(* PLC project Adressering.ecp, WAGO e!COCKPIT e!COCKPIT *)
(* stored: creationDateTime 2021-01-18T14:20:23.2110188, modificationDateTime 2021-01-18T11:51:27.6823754 *)

TYPE dtRomtype_22200000221102 : STRUCT
  RB601_V : BOOL;  (* Bevegelse *)
  RB602_V : BOOL;  (* Bevegelse *)
  RB601_HVAC : BOOL;  (* HVAC signal *)
  RB602_HVAC : BOOL;  (* HVAC signal *)
  RT601_CT : REAL;  (* Rom temperatur *)
  RT602_CT : REAL;  (* Rom temperatur *)
  RT602_SP : REAL;  (* Temperatur SP *)
  RT601_SP_D : REAL;  (* Temperatur SP *)
  RT601_SP_S : REAL;  (* Temperatur SP standby *)
  RT601_SP_N : REAL;  (* Temperatur SP nattsenk *)
  RT601_SP_F : REAL;  (* Temperatur SP frostsikring *)
  RT601_CS : REAL;  (* Aktivt temperatur SP *)
  OPM : INT;  (* Rom modus *)
  OPM_CV : INT;  (* Rom modus verdi *)
  RT601_SP : REAL;  (* Temperatur SP feedback *)
  RT601_SP_FB : REAL;  (* Temperatur SP *)
  RT601_SP_IN : REAL;  (* Temperatur SP lokalt panel *)
  RT602_SP_FB : REAL;  (* Temperatur SP *)
  RT602_SP_IN : REAL;  (* Temperatur SP lokalt panel *)
  LU601_V : BOOL;  (* Befukter status *)
  LU601_AL : BOOL;  (* Befukter alarm/feil *)
  OPM_001 : BYTE;  (* OPM output *)
  OPM_002 : BYTE;  (* OPM output *)
END_STRUCT;
END_TYPE

TYPE dtRomtype_1120011 : STRUCT
  RB601_V : BOOL;  (* Bevegelse *)
  RB601_HVAC : BOOL;  (* HVAC signal *)
  RT601_CT : REAL;  (* Rom temperatur *)
  RT602_CT : REAL;  (* Rom temperatur *)
  RT602_SP : REAL;  (* Temperatur SP *)
  RT601_SP_D : REAL;  (* Temperatur SP *)
  RT601_SP_S : REAL;  (* Temperatur SP standby *)
  RT601_SP_N : REAL;  (* Temperatur SP nattsenk *)
  RT601_SP_F : REAL;  (* Temperatur SP frostsikring *)
  RT601_CS : REAL;  (* Aktivt temperatur SP *)
  OPM : INT;  (* Rom modus *)
  OPM_CV : INT;  (* Rom modus verdi *)
  LH601_CMD : BOOL;  (* LH601_CMD *)
  LH601_MAN : BOOL;  (* Force LH *)
  LC601_OP : REAL;  (* LC601_OP *)
  LC601_SP : REAL;  (* LC SP *)
  LC601_MAN : BOOL;  (* Force LC *)
END_STRUCT;
END_TYPE

TYPE dtRomtype_112001 : STRUCT
  RB601_V : BOOL;  (* Bevegelse *)
  RB601_HVAC : BOOL;  (* HVAC signal *)
  RT601_CT : REAL;  (* Rom temperatur *)
  RT602_CT : REAL;  (* Rom temperatur *)
  RT602_SP : REAL;  (* Temperatur SP *)
  RT601_SP_D : REAL;  (* Temperatur SP *)
  RT601_SP_S : REAL;  (* Temperatur SP standby *)
  RT601_SP_N : REAL;  (* Temperatur SP nattsenk *)
  RT601_SP_F : REAL;  (* Temperatur SP frostsikring *)
  RT601_CS : REAL;  (* Aktivt temperatur SP *)
  OPM : INT;  (* Rom modus *)
  OPM_CV : INT;  (* Rom modus verdi *)
  LH601_CMD : BOOL;  (* LH601_CMD *)
  LH601_MAN : BOOL;  (* Force LH *)
END_STRUCT;
END_TYPE

TYPE dtRomtype_112101 : STRUCT
  RB601_V : BOOL;  (* Bevegelse *)
  RB601_HVAC : BOOL;  (* HVAC signal *)
  RT601_CT : REAL;  (* Rom temperatur *)
  RT602_CT : REAL;  (* Rom temperatur *)
  RT602_SP : REAL;  (* Temperatur SP *)
  RT601_SP_D : REAL;  (* Temperatur SP *)
  RT601_SP_S : REAL;  (* Temperatur SP standby *)
  RT601_SP_N : REAL;  (* Temperatur SP nattsenk *)
  RT601_SP_F : REAL;  (* Temperatur SP frostsikring *)
  RT601_CS : REAL;  (* Aktivt temperatur SP *)
  OPM : INT;  (* Rom modus *)
  OPM_CV : INT;  (* Rom modus verdi *)
  RY601_CV : REAL;  (* Co2 Nivaa *)
  RY601_SP : REAL;  (* Co2 SP *)
  RY601_OP : REAL;  (* Co2 paadrag *)
  LH601_CMD : BOOL;  (* LH601_CMD *)
  LH601_MAN : BOOL;  (* Force LH *)
END_STRUCT;
END_TYPE

TYPE dtRomtype_112002 : STRUCT
  RB601_V : BOOL;  (* Bevegelse *)
  RB601_HVAC : BOOL;  (* HVAC signal *)
  RT601_CT : REAL;  (* Rom temperatur *)
  RT602_CT : REAL;  (* Rom temperatur *)
  RT602_SP : REAL;  (* Temperatur SP *)
  RT601_SP_D : REAL;  (* Temperatur SP *)
  RT601_SP_S : REAL;  (* Temperatur SP standby *)
  RT601_SP_N : REAL;  (* Temperatur SP nattsenk *)
  RT601_SP_F : REAL;  (* Temperatur SP frostsikring *)
  RT601_CS : REAL;  (* Aktivt temperatur SP *)
  OPM : INT;  (* Rom modus *)
  OPM_CV : INT;  (* Rom modus verdi *)
  LH601_CMD : BOOL;  (* LH601_CMD *)
  LH602_CMD : BOOL;  (* LH602_CMD *)
  LH601_MAN : BOOL;  (* Force LH *)
END_STRUCT;
END_TYPE

TYPE dtRomtype_22 : STRUCT
  RB601_V : BOOL;  (* Bevegelse *)
  RB602_V : BOOL;  (* Bevegelse *)
  RB601_HVAC : BOOL;  (* HVAC signal *)
  RB602_HVAC : BOOL;  (* HVAC signal *)
END_STRUCT;
END_TYPE

TYPE dtRomtype_11 : STRUCT
  RB601_V : BOOL;  (* Bevegelse *)
  RB601_HVAC : BOOL;  (* HVAC signal *)
END_STRUCT;
END_TYPE

TYPE dtRomtype_4462051 : STRUCT
  RB601_V : BOOL;  (* Bevegelse *)
  RB602_V : BOOL;  (* Bevegelse *)
  RB603_V : BOOL;  (* Bevegelse *)
  RB604_V : BOOL;  (* Bevegelse *)
  RB601_HVAC : BOOL;  (* HVAC signal *)
  RB602_HVAC : BOOL;  (* HVAC signal *)
  RB603_HVAC : BOOL;  (* HVAC signal *)
  RB604_HVAC : BOOL;  (* HVAC signal *)
  RT601_CT : REAL;  (* Rom temperatur *)
  RT602_CT : REAL;  (* Rom temperatur *)
  RT602_SP : REAL;  (* Temperatur SP *)
  RT603_CT : REAL;  (* Rom temperatur *)
  RT603_SP : REAL;  (* Temperatur SP *)
  RT604_CT : REAL;  (* Rom temperatur *)
  RT604_SP : REAL;  (* Temperatur SP *)
  RT605_CT : REAL;  (* Rom temperatur *)
  RT605_SP : REAL;  (* Temperatur SP *)
  RT606_CT : REAL;  (* Rom temperatur *)
  RT606_SP : REAL;  (* Temperatur SP *)
  RT601_SP_D : REAL;  (* Temperatur SP *)
  RT601_SP_S : REAL;  (* Temperatur SP standby *)
  RT601_SP_N : REAL;  (* Temperatur SP nattsenk *)
  RT601_SP_F : REAL;  (* Temperatur SP frostsikring *)
  RT601_CS : REAL;  (* Aktivt temperatur SP *)
  OPM : INT;  (* Rom modus *)
  OPM_CV : INT;  (* Rom modus verdi *)
  RY601_CV : REAL;  (* Co2 Nivaa *)
  RY602_CV : REAL;  (* Co2 Nivaa *)
  RY601_SP : REAL;  (* Co2 SP *)
  RY601_OP : REAL;  (* Co2 paadrag *)
  LH601_CMD : BOOL;  (* LH601_CMD *)
  LH602_CMD : BOOL;  (* LH602_CMD *)
  LH603_CMD : BOOL;  (* LH603_CMD *)
  LH604_CMD : BOOL;  (* LH604_CMD *)
  LH605_CMD : BOOL;  (* LH605_CMD *)
  LH601_MAN : BOOL;  (* Force LH *)
  LC601_OP : REAL;  (* LC601_OP *)
  LC601_SP : REAL;  (* LC SP *)
  LC601_MAN : BOOL;  (* Force LC *)
END_STRUCT;
END_TYPE

TYPE dtRomtype_003 : STRUCT
  RT601_CT : REAL;  (* Rom temperatur *)
  RT602_CT : REAL;  (* Rom temperatur *)
  RT602_SP : REAL;  (* Temperatur SP *)
  RT603_CT : REAL;  (* Rom temperatur *)
  RT603_SP : REAL;  (* Temperatur SP *)
  RT601_SP_D : REAL;  (* Temperatur SP *)
  RT601_SP_S : REAL;  (* Temperatur SP standby *)
  RT601_SP_N : REAL;  (* Temperatur SP nattsenk *)
  RT601_SP_F : REAL;  (* Temperatur SP frostsikring *)
  RT601_CS : REAL;  (* Aktivt temperatur SP *)
  OPM : INT;  (* Rom modus *)
  OPM_CV : INT;  (* Rom modus verdi *)
END_STRUCT;
END_TYPE

TYPE dtRomtype_1121011 : STRUCT
  RB601_V : BOOL;  (* Bevegelse *)
  RB601_HVAC : BOOL;  (* HVAC signal *)
  RT601_CT : REAL;  (* Rom temperatur *)
  RT602_CT : REAL;  (* Rom temperatur *)
  RT602_SP : REAL;  (* Temperatur SP *)
  RT601_SP_D : REAL;  (* Temperatur SP *)
  RT601_SP_S : REAL;  (* Temperatur SP standby *)
  RT601_SP_N : REAL;  (* Temperatur SP nattsenk *)
  RT601_SP_F : REAL;  (* Temperatur SP frostsikring *)
  RT601_CS : REAL;  (* Aktivt temperatur SP *)
  OPM : INT;  (* Rom modus *)
  OPM_CV : INT;  (* Rom modus verdi *)
  RY601_CV : REAL;  (* Co2 Nivaa *)
  RY601_SP : REAL;  (* Co2 SP *)
  RY601_OP : REAL;  (* Co2 paadrag *)
  LH601_CMD : BOOL;  (* LH601_CMD *)
  LH601_MAN : BOOL;  (* Force LH *)
  LC601_OP : REAL;  (* LC601_OP *)
  LC601_SP : REAL;  (* LC SP *)
  LC601_MAN : BOOL;  (* Force LC *)
END_STRUCT;
END_TYPE

{attribute 'qualified_only'}
VAR_GLOBAL  (* STLV59_563 *)
  STLV59_A_563_RB001_HVAC : BOOL;  (* HVAC signal for PLS *)
  STLV59_A_563_KNX_Card_1_Status : BOOL;  (* KNX kort 1 status *)
  STLV59_A_563_001 : dtRomtype_22200000221102;  (* Ostelager *)
  STLV59_A_563_002 : dtRomtype_1120011;  (* Sosial sone *)
  STLV59_A_563_003 : dtRomtype_112001;  (* Jugendstue (Egentlig romtype 110001, men får temp fra rom 004) *)
  STLV59_A_563_004 : dtRomtype_112101;  (* Gang jugend *)
  STLV59_A_563_005 : dtRomtype_112001;  (* Kjøkken *)
  STLV59_A_563_006 : dtRomtype_112002;  (* Trenings rom *)
  STLV59_A_563_007 : dtRomtype_112001;  (* Garderobe 2 *)
  STLV59_A_563_008 : dtRomtype_112001;  (* Garderobe 1 *)
  STLV59_A_563_009 : dtRomtype_112001;  (* WC *)
  STLV59_A_563_010 : dtRomtype_112001;  (* WC *)
  STLV59_A_563_011 : dtRomtype_112001;  (* Garderobe *)
  STLV59_A_563_012 : dtRomtype_112001;  (* Entre *)
  STLV59_A_563_013 : dtRomtype_112001;  (* Bøttekott *)
  STLV59_A_563_014 : dtRomtype_22;  (* Teknisk rom *)
  STLV59_A_563_015 : dtRomtype_11;  (* Krypkjeller *)
  STLV59_A_563_016 : dtRomtype_11;  (* Teknisk rom tårn *)
  STLV59_A_563_017 : dtRomtype_112001;  (* Arkiv *)
  STLV59_A_563_101 : dtRomtype_112001;  (* Vindfang *)
  STLV59_A_563_102 : dtRomtype_112001;  (* Garderobe *)
  STLV59_A_563_103 : dtRomtype_4462051;  (* Storsal *)
  STLV59_A_563_109 : dtRomtype_112001;  (* Forrom WC *)
  STLV59_A_563_201 : dtRomtype_003;  (* Landskap *)
  STLV59_A_563_212 : dtRomtype_1121011;  (* Møterom 4 *)
  STLV59_A_563_213 : dtRomtype_1120011;  (* Stillerom *)
  STLV59_A_563_T1_U1 : dtRomtype_112001;  (* Trapp 1 U1 *)
  STLV59_A_563_T2_1 : dtRomtype_112001;  (* Trapp 2 1. etg. *)
  STLV59_A_563_T2_2 : dtRomtype_112001;  (* Trapp 2 2. etg. *)
END_VAR

FUNCTION_BLOCK fbRomtype_22200000221102
  VAR_INPUT
    RB601_HVAC : BOOL;
    RB602_HVAC : BOOL;
    RT601_CT : REAL;
    RT602_CT : REAL;
    RT602_SP : REAL;
    RT601_SP_D : REAL;
    RT601_SP_S : REAL;
    RT601_SP_N : REAL;
    RT601_SP_F : REAL;
    OPM : INT;
    RT601_SP_IN : REAL;
    RT602_SP_IN : REAL;
    LU601_V : BOOL;
  END_VAR
  VAR_OUTPUT
    OPM_CV : INT;
    RT601_CS : REAL;
    RT602_CS : REAL;
    OPM_001 : BYTE;
    OPM_002 : BYTE;
  END_VAR

(* CFC diagram, written out as Structured Text *)
END_FUNCTION_BLOCK

FUNCTION_BLOCK fbRomtype_1120011
  VAR_INPUT
    RB601_HVAC : BOOL;
    RT601_CT : REAL;
    RT602_CT : REAL;
    RT602_SP : REAL;
    RT601_SP_D : REAL;
    RT601_SP_S : REAL;
    RT601_SP_N : REAL;
    RT601_SP_F : REAL;
    OPM : INT;
    LH601_MAN : BOOL;
    LC601_SP : REAL;
    LC601_MAN : BOOL;
  END_VAR
  VAR_OUTPUT
    OPM_CV : INT;
    RT601_CS : REAL;
    RT602_CS : REAL;
    LH601_CMD : BOOL;
    LC601_OP : REAL;
  END_VAR

(* CFC diagram, written out as Structured Text *)
END_FUNCTION_BLOCK

FUNCTION_BLOCK fbRomtype_112001
  VAR_INPUT
    RB601_HVAC : BOOL;
    RT601_CT : REAL;
    RT602_CT : REAL;
    RT602_SP : REAL;
    RT601_SP_D : REAL;
    RT601_SP_S : REAL;
    RT601_SP_N : REAL;
    RT601_SP_F : REAL;
    OPM : INT;
    LH601_MAN : BOOL;
  END_VAR
  VAR_OUTPUT
    OPM_CV : INT;
    RT601_CS : REAL;
    RT602_CS : REAL;
    LH601_CMD : BOOL;
  END_VAR

(* CFC diagram, written out as Structured Text *)
END_FUNCTION_BLOCK

FUNCTION_BLOCK fbRomtype_112101
  VAR_INPUT
    RB601_HVAC : BOOL;
    RT601_CT : REAL;
    RT602_CT : REAL;
    RT602_SP : REAL;
    RT601_SP_D : REAL;
    RT601_SP_S : REAL;
    RT601_SP_N : REAL;
    RT601_SP_F : REAL;
    OPM : INT;
    RY601_CV : REAL;
    RY601_SP : REAL;
    LH601_MAN : BOOL;
  END_VAR
  VAR_OUTPUT
    OPM_CV : INT;
    RT601_CS : REAL;
    RT602_CS : REAL;
    RY601_OP : REAL;
    LH601_CMD : BOOL;
  END_VAR

(* CFC diagram, written out as Structured Text *)
END_FUNCTION_BLOCK

FUNCTION_BLOCK fbRomtype_112002
  VAR_INPUT
    RB601_HVAC : BOOL;
    RT601_CT : REAL;
    RT602_CT : REAL;
    RT602_SP : REAL;
    RT601_SP_D : REAL;
    RT601_SP_S : REAL;
    RT601_SP_N : REAL;
    RT601_SP_F : REAL;
    OPM : INT;
    LH601_MAN : BOOL;
  END_VAR
  VAR_OUTPUT
    OPM_CV : INT;
    RT601_CS : REAL;
    RT602_CS : REAL;
    LH601_CMD : BOOL;
    LH602_CMD : BOOL;
  END_VAR

(* CFC diagram, written out as Structured Text *)
END_FUNCTION_BLOCK

FUNCTION_BLOCK fbRomtype_4462051
  VAR_INPUT
    RB601_HVAC : BOOL;
    RB602_HVAC : BOOL;
    RB603_HVAC : BOOL;
    RB604_HVAC : BOOL;
    RT601_CT : REAL;
    RT602_CT : REAL;
    RT602_SP : REAL;
    RT603_CT : REAL;
    RT603_SP : REAL;
    RT604_CT : REAL;
    RT604_SP : REAL;
    RT605_CT : REAL;
    RT605_SP : REAL;
    RT606_CT : REAL;
    RT606_SP : REAL;
    RT601_SP_D : REAL;
    RT601_SP_S : REAL;
    RT601_SP_N : REAL;
    RT601_SP_F : REAL;
    OPM : INT;
    RY601_CV : REAL;
    RY602_CV : REAL;
    RY601_SP : REAL;
    LH601_MAN : BOOL;
    LC601_SP : REAL;
    LC601_MAN : BOOL;
  END_VAR
  VAR_OUTPUT
    OPM_CV : INT;
    RT601_CS : REAL;
    RT602_CS : REAL;
    RT603_CS : REAL;
    RT604_CS : REAL;
    RT605_CS : REAL;
    RT606_CS : REAL;
    RY601_OP : REAL;
    LH601_CMD : BOOL;
    LH602_CMD : BOOL;
    LH603_CMD : BOOL;
    LH604_CMD : BOOL;
    LH605_CMD : BOOL;
    LC601_OP : REAL;
  END_VAR

(* CFC diagram, written out as Structured Text *)
END_FUNCTION_BLOCK

FUNCTION_BLOCK fbRomtype_1121011
  VAR_INPUT
    RB601_HVAC : BOOL;
    RT601_CT : REAL;
    RT602_CT : REAL;
    RT602_SP : REAL;
    RT601_SP_D : REAL;
    RT601_SP_S : REAL;
    RT601_SP_N : REAL;
    RT601_SP_F : REAL;
    OPM : INT;
    RY601_CV : REAL;
    RY601_SP : REAL;
    LH601_MAN : BOOL;
    LC601_SP : REAL;
    LC601_MAN : BOOL;
  END_VAR
  VAR_OUTPUT
    OPM_CV : INT;
    RT601_CS : REAL;
    RT602_CS : REAL;
    RY601_OP : REAL;
    LH601_CMD : BOOL;
    LC601_OP : REAL;
  END_VAR

(* CFC diagram, written out as Structured Text *)
END_FUNCTION_BLOCK

PROGRAM PRG_KNX_563_1
  VAR
    i : INT := 0;  (* Felles *)
    Interval : OSCAT_BASIC.CLK_PRG;
    typDPT : typDPT;
    KNX_master_1 : WagoAppKNX.FbKNX_Master;  (* Master *)
    M1_001_001_RB601_V : fbDPT_Switch_pro;  (* 001 *)
    M1_002_001_RB602_V : fbDPT_Switch_pro;
    M1_003_001_RB601_HVAC : fbDPT_Switch_pro;
    M1_004_001_RB602_HVAC : fbDPT_Switch_pro;
    M1_005_001_RT601_SP : fbDPT_Value_Temp_pro;
    M1_006_001_RT602_SP : fbDPT_Value_Temp_pro;
    M1_007_001_RT601_SP_FB : fbDPT_Value_Temp_pro;
    M1_008_001_RT602_SP_FB : fbDPT_Value_Temp_pro;
    M1_009_001_OPM_001 : fbDPT_1_BYTE;
    M1_0010_001_OPM_002 : fbDPT_1_BYTE;
    M1_011_002_RB601_V : fbDPT_Switch_pro;  (* 002 *)
    M1_012_002_RB601_HVAC : fbDPT_Switch_pro;
    M1_013_002_RT601_CT : fbDPT_Value_Temp_pro;
    M1_014_002_RT602_CT : fbDPT_Value_Temp_pro;
    M1_015_003_RB601_V : fbDPT_Switch_pro;  (* 003 *)
    M1_016_003_RB601_HVAC : fbDPT_Switch_pro;
    M1_017_004_RB601_V : fbDPT_Switch_pro;  (* 004 *)
    M1_018_004_RB601_HVAC : fbDPT_Switch_pro;
    M1_019_004_RT601_CT : fbDPT_Value_Temp_pro;
    M1_020_004_RT602_CT : fbDPT_Value_Temp_pro;
    M1_021_004_RY601_CV : fbDPT_Value_AirQuality_pro;
    M1_022_005_RB601_V : fbDPT_Switch_pro;  (* 005 *)
    M1_023_005_RB601_HVAC : fbDPT_Switch_pro;
    M1_024_005_RT601_CT : fbDPT_Value_Temp_pro;
    M1_025_005_RT602_CT : fbDPT_Value_Temp_pro;
    M1_026_006_RB601_V : fbDPT_Switch_pro;  (* 006 *)
    M1_027_006_RB601_HVAC : fbDPT_Switch_pro;
    M1_028_006_RT601_CT : fbDPT_Value_Temp_pro;
    M1_029_007_RB601_V : fbDPT_Switch_pro;  (* 007 *)
    M1_030_007_RB601_HVAC : fbDPT_Switch_pro;
    M1_031_007_RT601_CT : fbDPT_Value_Temp_pro;
    M1_032_007_RT602_CT : fbDPT_Value_Temp_pro;
    M1_033_008_RB601_V : fbDPT_Switch_pro;  (* 008 *)
    M1_034_008_RB601_HVAC : fbDPT_Switch_pro;
    M1_035_008_RT601_CT : fbDPT_Value_Temp_pro;
    M1_036_008_RT602_CT : fbDPT_Value_Temp_pro;
    M1_037_009_RB601_V : fbDPT_Switch_pro;  (* 009 *)
    M1_038_009_RB601_HVAC : fbDPT_Switch_pro;
    M1_039_009_RT601_CT : fbDPT_Value_Temp_pro;
    M1_040_009_RT602_CT : fbDPT_Value_Temp_pro;
    M1_041_010_RB601_V : fbDPT_Switch_pro;  (* 010 *)
    M1_042_010_RB601_HVAC : fbDPT_Switch_pro;
    M1_043_010_RT601_CT : fbDPT_Value_Temp_pro;
    M1_044_010_RT602_CT : fbDPT_Value_Temp_pro;
    M1_045_011_RB601_V : fbDPT_Switch_pro;  (* 011 *)
    M1_046_011_RB601_HVAC : fbDPT_Switch_pro;
    M1_047_011_RT601_CT : fbDPT_Value_Temp_pro;
    M1_048_011_RT602_CT : fbDPT_Value_Temp_pro;
    M1_049_012_RB601_V : fbDPT_Switch_pro;  (* 012 *)
    M1_050_012_RB601_HVAC : fbDPT_Switch_pro;
    M1_051_012_RT601_CT : fbDPT_Value_Temp_pro;
    M1_052_012_RT602_CT : fbDPT_Value_Temp_pro;
    M1_053_013_RB601_V : fbDPT_Switch_pro;  (* 013 *)
    M1_054_013_RB601_HVAC : fbDPT_Switch_pro;
    M1_055_013_RT601_CT : fbDPT_Value_Temp_pro;
    M1_056_013_RT602_CT : fbDPT_Value_Temp_pro;
    M1_057_014_RB601_V : fbDPT_Switch_pro;  (* 014 *)
    M1_058_014_RB602_V : fbDPT_Switch_pro;
    M1_059_014_RB601_HVAC : fbDPT_Switch_pro;
    M1_060_014_RB602_HVAC : fbDPT_Switch_pro;
    M1_061_015_RB601_V : fbDPT_Switch_pro;  (* 015 *)
    M1_062_015_RB601_HVAC : fbDPT_Switch_pro;
    M1_063_016_RB601_V : fbDPT_Switch_pro;  (* 016 *)
    M1_064_016_RB601_HVAC : fbDPT_Switch_pro;
    M1_065_017_RB601_V : fbDPT_Switch_pro;  (* 017 *)
    M1_066_017_RB601_HVAC : fbDPT_Switch_pro;
    M1_067_017_RT601_CT : fbDPT_Value_Temp_pro;
    M1_068_017_RT602_CT : fbDPT_Value_Temp_pro;
    M1_069_101_RB601_V : fbDPT_Switch_pro;  (* 101 *)
    M1_070_101_RB601_HVAC : fbDPT_Switch_pro;
    M1_071_101_RT601_CT : fbDPT_Value_Temp_pro;
    M1_072_101_RT602_CT : fbDPT_Value_Temp_pro;
    M1_073_102_RB601_V : fbDPT_Switch_pro;  (* 102 *)
    M1_074_102_RB601_HVAC : fbDPT_Switch_pro;
    M1_075_102_RT601_CT : fbDPT_Value_Temp_pro;
    M1_076_102_RT602_CT : fbDPT_Value_Temp_pro;
    M1_077_103_RB601_V : fbDPT_Switch_pro;  (* 103 *)
    M1_078_103_RB602_V : fbDPT_Switch_pro;
    M1_079_103_RB603_V : fbDPT_Switch_pro;
    M1_080_103_RB604_V : fbDPT_Switch_pro;
    M1_081_103_RB601_HVAC : fbDPT_Switch_pro;
    M1_082_103_RB602_HVAC : fbDPT_Switch_pro;
    M1_083_103_RB603_HVAC : fbDPT_Switch_pro;
    M1_084_103_RB604_HVAC : fbDPT_Switch_pro;
    M1_085_103_RT601_CT : fbDPT_Value_Temp_pro;
    M1_086_103_RT602_CT : fbDPT_Value_Temp_pro;
    M1_087_103_RT603_CT : fbDPT_Value_Temp_pro;
    M1_088_103_RT604_CT : fbDPT_Value_Temp_pro;
    M1_089_109_RB601_V : fbDPT_Switch_pro;  (* 109 *)
    M1_090_109_RB601_HVAC : fbDPT_Switch_pro;
    M1_091_109_RT601_CT : fbDPT_Value_Temp_pro;
    M1_092_109_RT602_CT : fbDPT_Value_Temp_pro;
    M1_093_201_RT601_CT : fbDPT_Value_Temp_pro;  (* 201 *)
    M1_094_201_RT602_CT : fbDPT_Value_Temp_pro;
    M1_095_201_RT603_CT : fbDPT_Value_Temp_pro;
    M1_096_212_RB601_V : fbDPT_Switch_pro;  (* 212 *)
    M1_097_212_RB601_HVAC : fbDPT_Switch_pro;
    M1_098_212_RT601_CT : fbDPT_Value_Temp_pro;
    M1_099_212_RT602_CT : fbDPT_Value_Temp_pro;
    M1_100_212_RY601_CV : fbDPT_Value_AirQuality_pro;
    M1_101_213_RB601_V : fbDPT_Switch_pro;  (* 213 *)
    M1_102_213_RB601_HVAC : fbDPT_Switch_pro;
    M1_103_213_RT601_CT : fbDPT_Value_Temp_pro;
    M1_104_213_RT602_CT : fbDPT_Value_Temp_pro;
    M1_105_T1_U1_RB601_V : fbDPT_Switch_pro;  (* T1_U1 *)
    M1_106_T1_U1_RB601_HVAC : fbDPT_Switch_pro;
    M1_107_T1_U1_RT601_CT : fbDPT_Value_Temp_pro;
    M1_108_T1_U1_RT602_CT : fbDPT_Value_Temp_pro;
    M1_109_T2_1_RB601_V : fbDPT_Switch_pro;  (* T2_1 *)
    M1_110_T2_1_RB601_HVAC : fbDPT_Switch_pro;
    M1_111_T2_1_RT601_CT : fbDPT_Value_Temp_pro;
    M1_112_T2_1_RT602_CT : fbDPT_Value_Temp_pro;
    M1_113_T2_2_RB601_V : fbDPT_Switch_pro;  (* T2_2 *)
    M1_114_T2_2_RB601_HVAC : fbDPT_Switch_pro;
    M1_115_T2_2_RT601_CT : fbDPT_Value_Temp_pro;
    M1_116_T2_2_RT602_CT : fbDPT_Value_Temp_pro;
  END_VAR
  VAR  (* added by the conversion: wires and edge detectors of the diagram *)
    _ADD9_OUT : INT;
    _GT15_OUT : BOOL;
    _MOVE19_ENO : BOOL;
    _MOVE19_OUT : INT;
  END_VAR

(* CFC diagram, written out as Structured Text *)
(* KNX Sending interval *)
(* KNX Master *)
Interval(PT := t#2M);
_ADD9_OUT := BOOL_TO_INT(Interval.Q) + i;
i := _ADD9_OUT;
_GT15_OUT := i > 0;
_MOVE19_OUT := MOVE(EN := _GT15_OUT, IN := 0, ENO => _MOVE19_ENO);
IF _MOVE19_ENO THEN i := _MOVE19_OUT; END_IF;
KNX_master_1(I_Port := IoConfig_Globals.KNX_EIB_TP1_Interface, bPortKNX := 1);
STLV59_563.STLV59_A_563_KNX_Card_1_Status := KNX_master_1.sStatus = 'OK';
(* Rom 001 *)
(* RB601_V *)
(* RB602_V *)
M1_001_001_RB601_V(bPortKNX := 1, dwIndex_DPT := 1, typDPT := typDPT);
STLV59_563.STLV59_A_563_001.RB601_V := M1_001_001_RB601_V.xSwitch_OUT;
M1_002_001_RB602_V(bPortKNX := 1, dwIndex_DPT := 2, typDPT := typDPT);
STLV59_563.STLV59_A_563_001.RB602_V := M1_002_001_RB602_V.xSwitch_OUT;
(* RB601_HVAC *)
(* RB602_HVAC *)
M1_003_001_RB601_HVAC(bPortKNX := 1, dwIndex_DPT := 3, typDPT := typDPT);
STLV59_563.STLV59_A_563_001.RB601_HVAC := M1_003_001_RB601_HVAC.xSwitch_OUT;
M1_004_001_RB602_HVAC(bPortKNX := 1, dwIndex_DPT := 4, typDPT := typDPT);
STLV59_563.STLV59_A_563_001.RB602_HVAC := M1_004_001_RB602_HVAC.xSwitch_OUT;
(* RT601_SP *)
(* RT602_SP *)
M1_005_001_RT601_SP(bPortKNX := 1, dwIndex_DPT := 5, rValue_IN := STLV59_563.STLV59_A_563_001.RT601_SP_D, xUpdate_KNX := NOT STLV59_563.STLV59_A_563_001.RB601_HVAC, typDPT := typDPT);
M1_006_001_RT602_SP(bPortKNX := 1, dwIndex_DPT := 6, rValue_IN := STLV59_563.STLV59_A_563_001.RT602_SP, xUpdate_KNX := NOT STLV59_563.STLV59_A_563_001.RB601_HVAC, typDPT := typDPT);
(* RT601_SP Feedback *)
(* RT602_SP Feedback *)
M1_007_001_RT601_SP_FB(bPortKNX := 1, dwIndex_DPT := 7, typDPT := typDPT);
STLV59_563.STLV59_A_563_001.RT601_SP_IN := M1_007_001_RT601_SP_FB.rValue_OUT;
M1_008_001_RT602_SP_FB(bPortKNX := 1, dwIndex_DPT := 8, typDPT := typDPT);
STLV59_563.STLV59_A_563_001.RT602_SP_IN := M1_008_001_RT602_SP_FB.rValue_OUT;
(* OPM_001 *)
(* OPM_002 *)
M1_009_001_OPM_001(bPortKNX := 1, dwIndex_DPT := 9, bIN := STLV59_563.STLV59_A_563_001.OPM_001, xUpdate_KNX := i = 0, typDPT := typDPT);
M1_0010_001_OPM_002(bPortKNX := 1, dwIndex_DPT := 10, bIN := STLV59_563.STLV59_A_563_001.OPM_002, xUpdate_KNX := i = 1, typDPT := typDPT);
(* Rom 002 *)
(* RB601_V *)
(* RB601_HVAC *)
M1_011_002_RB601_V(bPortKNX := 1, dwIndex_DPT := 11, typDPT := typDPT);
STLV59_563.STLV59_A_563_002.RB601_V := M1_011_002_RB601_V.xSwitch_OUT;
M1_012_002_RB601_HVAC(bPortKNX := 1, dwIndex_DPT := 12, typDPT := typDPT);
STLV59_563.STLV59_A_563_002.RB601_HVAC := M1_012_002_RB601_HVAC.xSwitch_OUT;
(* RT601_CT *)
(* RT602_CT *)
M1_013_002_RT601_CT(bPortKNX := 1, dwIndex_DPT := 13, typDPT := typDPT);
STLV59_563.STLV59_A_563_002.RT601_CT := M1_013_002_RT601_CT.rValue_OUT;
M1_014_002_RT602_CT(bPortKNX := 1, dwIndex_DPT := 14, typDPT := typDPT);
STLV59_563.STLV59_A_563_002.RT602_CT := M1_014_002_RT602_CT.rValue_OUT;
(* Rom 003 *)
(* RB601_V *)
(* RB601_HVAC *)
M1_015_003_RB601_V(bPortKNX := 1, dwIndex_DPT := 15, typDPT := typDPT);
STLV59_563.STLV59_A_563_003.RB601_V := M1_015_003_RB601_V.xSwitch_OUT;
M1_016_003_RB601_HVAC(bPortKNX := 1, dwIndex_DPT := 16, typDPT := typDPT);
STLV59_563.STLV59_A_563_003.RB601_HVAC := M1_016_003_RB601_HVAC.xSwitch_OUT;
(* Rom 004 *)
(* RB601_V *)
(* RB601_HVAC *)
M1_017_004_RB601_V(bPortKNX := 1, dwIndex_DPT := 17, typDPT := typDPT);
STLV59_563.STLV59_A_563_004.RB601_V := M1_017_004_RB601_V.xSwitch_OUT;
M1_018_004_RB601_HVAC(bPortKNX := 1, dwIndex_DPT := 18, typDPT := typDPT);
STLV59_563.STLV59_A_563_004.RB601_HVAC := M1_018_004_RB601_HVAC.xSwitch_OUT;
(* RT601_CT *)
(* RT602_CT *)
M1_019_004_RT601_CT(bPortKNX := 1, dwIndex_DPT := 19, typDPT := typDPT);
STLV59_563.STLV59_A_563_004.RT601_CT := M1_019_004_RT601_CT.rValue_OUT;
M1_020_004_RT602_CT(bPortKNX := 1, dwIndex_DPT := 20, typDPT := typDPT);
STLV59_563.STLV59_A_563_004.RT602_CT := M1_020_004_RT602_CT.rValue_OUT;
(* RY601_CV *)
M1_021_004_RY601_CV(bPortKNX := 1, dwIndex_DPT := 21, typDPT := typDPT);
STLV59_563.STLV59_A_563_004.RY601_CV := M1_021_004_RY601_CV.rValue_OUT;
(* Rom 005 *)
(* RB601_V *)
(* RB601_HVAC *)
M1_022_005_RB601_V(bPortKNX := 1, dwIndex_DPT := 22, typDPT := typDPT);
STLV59_563.STLV59_A_563_005.RB601_V := M1_022_005_RB601_V.xSwitch_OUT;
M1_023_005_RB601_HVAC(bPortKNX := 1, dwIndex_DPT := 23, typDPT := typDPT);
STLV59_563.STLV59_A_563_005.RB601_HVAC := M1_023_005_RB601_HVAC.xSwitch_OUT;
(* RT601_CT *)
(* RT602_CT *)
M1_024_005_RT601_CT(bPortKNX := 1, dwIndex_DPT := 24, typDPT := typDPT);
STLV59_563.STLV59_A_563_005.RT601_CT := M1_024_005_RT601_CT.rValue_OUT;
M1_025_005_RT602_CT(bPortKNX := 1, dwIndex_DPT := 25, typDPT := typDPT);
STLV59_563.STLV59_A_563_005.RT602_CT := M1_025_005_RT602_CT.rValue_OUT;
(* Rom 006 *)
(* RB601_V *)
(* RB601_HVAC *)
M1_026_006_RB601_V(bPortKNX := 1, dwIndex_DPT := 26, typDPT := typDPT);
STLV59_563.STLV59_A_563_006.RB601_V := M1_026_006_RB601_V.xSwitch_OUT;
M1_027_006_RB601_HVAC(bPortKNX := 1, dwIndex_DPT := 27, typDPT := typDPT);
STLV59_563.STLV59_A_563_006.RB601_HVAC := M1_027_006_RB601_HVAC.xSwitch_OUT;
(* RT601_CT *)
M1_028_006_RT601_CT(bPortKNX := 1, dwIndex_DPT := 28, typDPT := typDPT);
STLV59_563.STLV59_A_563_006.RT601_CT := M1_028_006_RT601_CT.rValue_OUT;
(* Rom 007 *)
(* RB601_V *)
(* RB601_HVAC *)
M1_029_007_RB601_V(bPortKNX := 1, dwIndex_DPT := 29, typDPT := typDPT);
STLV59_563.STLV59_A_563_007.RB601_V := M1_029_007_RB601_V.xSwitch_OUT;
M1_030_007_RB601_HVAC(bPortKNX := 1, dwIndex_DPT := 30, typDPT := typDPT);
STLV59_563.STLV59_A_563_007.RB601_HVAC := M1_030_007_RB601_HVAC.xSwitch_OUT;
(* RT601_CT *)
(* RT602_CT *)
M1_031_007_RT601_CT(bPortKNX := 1, dwIndex_DPT := 31, typDPT := typDPT);
STLV59_563.STLV59_A_563_007.RT601_CT := M1_031_007_RT601_CT.rValue_OUT;
M1_032_007_RT602_CT(bPortKNX := 1, dwIndex_DPT := 32, typDPT := typDPT);
STLV59_563.STLV59_A_563_007.RT602_CT := M1_032_007_RT602_CT.rValue_OUT;
(* Rom 008 *)
(* RB601_V *)
(* RB601_HVAC *)
M1_033_008_RB601_V(bPortKNX := 1, dwIndex_DPT := 33, typDPT := typDPT);
STLV59_563.STLV59_A_563_008.RB601_V := M1_033_008_RB601_V.xSwitch_OUT;
M1_034_008_RB601_HVAC(bPortKNX := 1, dwIndex_DPT := 34, typDPT := typDPT);
STLV59_563.STLV59_A_563_008.RB601_HVAC := M1_034_008_RB601_HVAC.xSwitch_OUT;
(* RT601_CT *)
(* RT602_CT *)
M1_035_008_RT601_CT(bPortKNX := 1, dwIndex_DPT := 35, typDPT := typDPT);
STLV59_563.STLV59_A_563_008.RT601_CT := M1_035_008_RT601_CT.rValue_OUT;
M1_036_008_RT602_CT(bPortKNX := 1, dwIndex_DPT := 36, typDPT := typDPT);
STLV59_563.STLV59_A_563_008.RT602_CT := M1_036_008_RT602_CT.rValue_OUT;
(* Rom 009 *)
(* RB601_V *)
(* RB601_HVAC *)
M1_037_009_RB601_V(bPortKNX := 1, dwIndex_DPT := 37, typDPT := typDPT);
STLV59_563.STLV59_A_563_009.RB601_V := M1_037_009_RB601_V.xSwitch_OUT;
M1_038_009_RB601_HVAC(bPortKNX := 1, dwIndex_DPT := 38, typDPT := typDPT);
STLV59_563.STLV59_A_563_009.RB601_HVAC := M1_038_009_RB601_HVAC.xSwitch_OUT;
(* RT601_CT *)
(* RT602_CT *)
M1_039_009_RT601_CT(bPortKNX := 1, dwIndex_DPT := 39, typDPT := typDPT);
STLV59_563.STLV59_A_563_009.RT601_CT := M1_039_009_RT601_CT.rValue_OUT;
M1_040_009_RT602_CT(bPortKNX := 1, dwIndex_DPT := 40, typDPT := typDPT);
STLV59_563.STLV59_A_563_009.RT602_CT := M1_040_009_RT602_CT.rValue_OUT;
(* Rom 010 *)
(* RB601_V *)
(* RB601_HVAC *)
M1_041_010_RB601_V(bPortKNX := 1, dwIndex_DPT := 41, typDPT := typDPT);
STLV59_563.STLV59_A_563_010.RB601_V := M1_041_010_RB601_V.xSwitch_OUT;
M1_042_010_RB601_HVAC(bPortKNX := 1, dwIndex_DPT := 42, typDPT := typDPT);
STLV59_563.STLV59_A_563_010.RB601_HVAC := M1_042_010_RB601_HVAC.xSwitch_OUT;
(* RT601_CT *)
(* RT602_CT *)
M1_043_010_RT601_CT(bPortKNX := 1, dwIndex_DPT := 43, typDPT := typDPT);
STLV59_563.STLV59_A_563_010.RT601_CT := M1_043_010_RT601_CT.rValue_OUT;
M1_044_010_RT602_CT(bPortKNX := 1, dwIndex_DPT := 44, typDPT := typDPT);
STLV59_563.STLV59_A_563_010.RT602_CT := M1_044_010_RT602_CT.rValue_OUT;
(* Rom 011 *)
(* RB601_V *)
(* RB601_HVAC *)
M1_045_011_RB601_V(bPortKNX := 1, dwIndex_DPT := 45, typDPT := typDPT);
STLV59_563.STLV59_A_563_011.RB601_V := M1_045_011_RB601_V.xSwitch_OUT;
M1_046_011_RB601_HVAC(bPortKNX := 1, dwIndex_DPT := 46, typDPT := typDPT);
STLV59_563.STLV59_A_563_011.RB601_HVAC := M1_046_011_RB601_HVAC.xSwitch_OUT;
(* RT601_CT *)
(* RT602_CT *)
M1_047_011_RT601_CT(bPortKNX := 1, dwIndex_DPT := 47, typDPT := typDPT);
STLV59_563.STLV59_A_563_011.RT601_CT := M1_047_011_RT601_CT.rValue_OUT;
M1_048_011_RT602_CT(bPortKNX := 1, dwIndex_DPT := 48, typDPT := typDPT);
STLV59_563.STLV59_A_563_011.RT602_CT := M1_048_011_RT602_CT.rValue_OUT;
(* Rom 012 *)
(* RB601_V *)
(* RB601_HVAC *)
M1_049_012_RB601_V(bPortKNX := 1, dwIndex_DPT := 49, typDPT := typDPT);
STLV59_563.STLV59_A_563_012.RB601_V := M1_049_012_RB601_V.xSwitch_OUT;
M1_050_012_RB601_HVAC(bPortKNX := 1, dwIndex_DPT := 50, typDPT := typDPT);
STLV59_563.STLV59_A_563_012.RB601_HVAC := M1_050_012_RB601_HVAC.xSwitch_OUT;
(* RT601_CT *)
(* RT602_CT *)
M1_051_012_RT601_CT(bPortKNX := 1, dwIndex_DPT := 51, typDPT := typDPT);
STLV59_563.STLV59_A_563_012.RT601_CT := M1_051_012_RT601_CT.rValue_OUT;
M1_052_012_RT602_CT(bPortKNX := 1, dwIndex_DPT := 52, typDPT := typDPT);
STLV59_563.STLV59_A_563_012.RT602_CT := M1_052_012_RT602_CT.rValue_OUT;
(* Rom 013 *)
(* RB601_V *)
(* RB601_HVAC *)
M1_053_013_RB601_V(bPortKNX := 1, dwIndex_DPT := 53, typDPT := typDPT);
STLV59_563.STLV59_A_563_013.RB601_V := M1_053_013_RB601_V.xSwitch_OUT;
M1_054_013_RB601_HVAC(bPortKNX := 1, dwIndex_DPT := 54, typDPT := typDPT);
STLV59_563.STLV59_A_563_013.RB601_HVAC := M1_054_013_RB601_HVAC.xSwitch_OUT;
(* RT601_CT *)
(* RT602_CT *)
M1_055_013_RT601_CT(bPortKNX := 1, dwIndex_DPT := 55, typDPT := typDPT);
STLV59_563.STLV59_A_563_013.RT601_CT := M1_055_013_RT601_CT.rValue_OUT;
M1_056_013_RT602_CT(bPortKNX := 1, dwIndex_DPT := 56, typDPT := typDPT);
STLV59_563.STLV59_A_563_013.RT602_CT := M1_056_013_RT602_CT.rValue_OUT;
(* Rom 014 *)
(* RB601_V *)
(* RB602_V *)
M1_057_014_RB601_V(bPortKNX := 1, dwIndex_DPT := 57, typDPT := typDPT);
STLV59_563.STLV59_A_563_014.RB601_V := M1_057_014_RB601_V.xSwitch_OUT;
M1_058_014_RB602_V(bPortKNX := 1, dwIndex_DPT := 58, typDPT := typDPT);
STLV59_563.STLV59_A_563_014.RB602_V := M1_058_014_RB602_V.xSwitch_OUT;
(* RB601_HVAC *)
(* RB602_HVAC *)
M1_059_014_RB601_HVAC(bPortKNX := 1, dwIndex_DPT := 59, typDPT := typDPT);
STLV59_563.STLV59_A_563_014.RB601_HVAC := M1_059_014_RB601_HVAC.xSwitch_OUT;
M1_060_014_RB602_HVAC(bPortKNX := 1, dwIndex_DPT := 60, typDPT := typDPT);
STLV59_563.STLV59_A_563_014.RB602_HVAC := M1_060_014_RB602_HVAC.xSwitch_OUT;
(* Rom 015 *)
(* RB601_V *)
(* RB601_HVAC *)
M1_061_015_RB601_V(bPortKNX := 1, dwIndex_DPT := 61, typDPT := typDPT);
STLV59_563.STLV59_A_563_015.RB601_V := M1_061_015_RB601_V.xSwitch_OUT;
M1_062_015_RB601_HVAC(bPortKNX := 1, dwIndex_DPT := 62, typDPT := typDPT);
STLV59_563.STLV59_A_563_015.RB601_HVAC := M1_062_015_RB601_HVAC.xSwitch_OUT;
(* Rom 016 *)
(* RB601_V *)
(* RB601_HVAC *)
M1_063_016_RB601_V(bPortKNX := 1, dwIndex_DPT := 63, typDPT := typDPT);
STLV59_563.STLV59_A_563_016.RB601_V := M1_063_016_RB601_V.xSwitch_OUT;
M1_064_016_RB601_HVAC(bPortKNX := 1, dwIndex_DPT := 64, typDPT := typDPT);
STLV59_563.STLV59_A_563_016.RB601_HVAC := M1_064_016_RB601_HVAC.xSwitch_OUT;
(* Rom 017 *)
(* RB601_V *)
(* RB601_HVAC *)
M1_065_017_RB601_V(bPortKNX := 1, dwIndex_DPT := 65, typDPT := typDPT);
STLV59_563.STLV59_A_563_017.RB601_V := M1_065_017_RB601_V.xSwitch_OUT;
M1_066_017_RB601_HVAC(bPortKNX := 1, dwIndex_DPT := 66, typDPT := typDPT);
STLV59_563.STLV59_A_563_017.RB601_HVAC := M1_066_017_RB601_HVAC.xSwitch_OUT;
(* RT601_CT *)
(* RT602_CT *)
M1_067_017_RT601_CT(bPortKNX := 1, dwIndex_DPT := 67, typDPT := typDPT);
STLV59_563.STLV59_A_563_017.RT601_CT := M1_067_017_RT601_CT.rValue_OUT;
M1_068_017_RT602_CT(bPortKNX := 1, dwIndex_DPT := 68, typDPT := typDPT);
STLV59_563.STLV59_A_563_017.RT602_CT := M1_068_017_RT602_CT.rValue_OUT;
(* Rom 101 *)
(* RB601_V *)
(* RB601_HVAC *)
M1_069_101_RB601_V(bPortKNX := 1, dwIndex_DPT := 69, typDPT := typDPT);
STLV59_563.STLV59_A_563_101.RB601_V := M1_069_101_RB601_V.xSwitch_OUT;
M1_070_101_RB601_HVAC(bPortKNX := 1, dwIndex_DPT := 70, typDPT := typDPT);
STLV59_563.STLV59_A_563_101.RB601_HVAC := M1_070_101_RB601_HVAC.xSwitch_OUT;
(* RT601_CT *)
(* RT602_CT *)
M1_071_101_RT601_CT(bPortKNX := 1, dwIndex_DPT := 71, typDPT := typDPT);
STLV59_563.STLV59_A_563_101.RT601_CT := M1_071_101_RT601_CT.rValue_OUT;
M1_072_101_RT602_CT(bPortKNX := 1, dwIndex_DPT := 72, typDPT := typDPT);
STLV59_563.STLV59_A_563_101.RT602_CT := M1_072_101_RT602_CT.rValue_OUT;
(* Rom 102 *)
(* RB601_V *)
(* RB601_HVAC *)
M1_073_102_RB601_V(bPortKNX := 1, dwIndex_DPT := 73, typDPT := typDPT);
STLV59_563.STLV59_A_563_102.RB601_V := M1_073_102_RB601_V.xSwitch_OUT;
M1_074_102_RB601_HVAC(bPortKNX := 1, dwIndex_DPT := 74, typDPT := typDPT);
STLV59_563.STLV59_A_563_102.RB601_HVAC := M1_074_102_RB601_HVAC.xSwitch_OUT;
(* RT601_CT *)
(* RT602_CT *)
M1_075_102_RT601_CT(bPortKNX := 1, dwIndex_DPT := 75, typDPT := typDPT);
STLV59_563.STLV59_A_563_102.RT601_CT := M1_075_102_RT601_CT.rValue_OUT;
M1_076_102_RT602_CT(bPortKNX := 1, dwIndex_DPT := 76, typDPT := typDPT);
STLV59_563.STLV59_A_563_102.RT602_CT := M1_076_102_RT602_CT.rValue_OUT;
(* Rom 103 *)
(* RB601_V *)
(* RB602_V *)
M1_077_103_RB601_V(bPortKNX := 1, dwIndex_DPT := 77, typDPT := typDPT);
STLV59_563.STLV59_A_563_103.RB601_V := M1_077_103_RB601_V.xSwitch_OUT;
M1_078_103_RB602_V(bPortKNX := 1, dwIndex_DPT := 78, typDPT := typDPT);
STLV59_563.STLV59_A_563_103.RB602_V := M1_078_103_RB602_V.xSwitch_OUT;
(* RB603_V *)
(* RB604_V *)
M1_079_103_RB603_V(bPortKNX := 1, dwIndex_DPT := 79, typDPT := typDPT);
STLV59_563.STLV59_A_563_103.RB603_V := M1_079_103_RB603_V.xSwitch_OUT;
M1_080_103_RB604_V(bPortKNX := 1, dwIndex_DPT := 80, typDPT := typDPT);
STLV59_563.STLV59_A_563_103.RB604_V := M1_080_103_RB604_V.xSwitch_OUT;
(* RB601_HVAC *)
(* RB602_HVAC *)
M1_081_103_RB601_HVAC(bPortKNX := 1, dwIndex_DPT := 81, typDPT := typDPT);
STLV59_563.STLV59_A_563_103.RB601_HVAC := M1_081_103_RB601_HVAC.xSwitch_OUT;
M1_082_103_RB602_HVAC(bPortKNX := 1, dwIndex_DPT := 82, typDPT := typDPT);
STLV59_563.STLV59_A_563_103.RB602_HVAC := M1_082_103_RB602_HVAC.xSwitch_OUT;
(* RB603_HVAC *)
(* RB604_HVAC *)
M1_083_103_RB603_HVAC(bPortKNX := 1, dwIndex_DPT := 83, typDPT := typDPT);
STLV59_563.STLV59_A_563_103.RB603_HVAC := M1_083_103_RB603_HVAC.xSwitch_OUT;
M1_084_103_RB604_HVAC(bPortKNX := 1, dwIndex_DPT := 84, typDPT := typDPT);
STLV59_563.STLV59_A_563_103.RB604_HVAC := M1_084_103_RB604_HVAC.xSwitch_OUT;
(* RT601_CT *)
(* RT602_CT *)
M1_085_103_RT601_CT(bPortKNX := 1, dwIndex_DPT := 85, typDPT := typDPT);
STLV59_563.STLV59_A_563_103.RT601_CT := M1_085_103_RT601_CT.rValue_OUT;
M1_086_103_RT602_CT(bPortKNX := 1, dwIndex_DPT := 86, typDPT := typDPT);
STLV59_563.STLV59_A_563_103.RT602_CT := M1_086_103_RT602_CT.rValue_OUT;
(* RT603_CT *)
(* RT604_CT *)
M1_087_103_RT603_CT(bPortKNX := 1, dwIndex_DPT := 87, typDPT := typDPT);
STLV59_563.STLV59_A_563_103.RT603_CT := M1_087_103_RT603_CT.rValue_OUT;
M1_088_103_RT604_CT(bPortKNX := 1, dwIndex_DPT := 88, typDPT := typDPT);
STLV59_563.STLV59_A_563_103.RT604_CT := M1_088_103_RT604_CT.rValue_OUT;
(* Rom 109 *)
(* RB601_V *)
(* RB601_HVAC *)
M1_089_109_RB601_V(bPortKNX := 1, dwIndex_DPT := 89, typDPT := typDPT);
STLV59_563.STLV59_A_563_109.RB601_V := M1_089_109_RB601_V.xSwitch_OUT;
M1_090_109_RB601_HVAC(bPortKNX := 1, dwIndex_DPT := 90, typDPT := typDPT);
STLV59_563.STLV59_A_563_109.RB601_HVAC := M1_090_109_RB601_HVAC.xSwitch_OUT;
(* RT601_CT *)
(* RT602_CT *)
M1_091_109_RT601_CT(bPortKNX := 1, dwIndex_DPT := 91, typDPT := typDPT);
STLV59_563.STLV59_A_563_109.RT601_CT := M1_091_109_RT601_CT.rValue_OUT;
M1_092_109_RT602_CT(bPortKNX := 1, dwIndex_DPT := 92, typDPT := typDPT);
STLV59_563.STLV59_A_563_109.RT602_CT := M1_092_109_RT602_CT.rValue_OUT;
(* Rom 201 *)
(* RT601_CT *)
(* RT602_CT *)
M1_093_201_RT601_CT(bPortKNX := 1, dwIndex_DPT := 93, typDPT := typDPT);
STLV59_563.STLV59_A_563_201.RT601_CT := M1_093_201_RT601_CT.rValue_OUT;
M1_094_201_RT602_CT(bPortKNX := 1, dwIndex_DPT := 94, typDPT := typDPT);
STLV59_563.STLV59_A_563_201.RT602_CT := M1_094_201_RT602_CT.rValue_OUT;
(* RT603_CT *)
M1_095_201_RT603_CT(bPortKNX := 1, dwIndex_DPT := 95, typDPT := typDPT);
STLV59_563.STLV59_A_563_201.RT603_CT := M1_095_201_RT603_CT.rValue_OUT;
(* Rom 212 *)
(* RB601_V *)
(* RB601_HVAC *)
M1_096_212_RB601_V(bPortKNX := 1, dwIndex_DPT := 96, typDPT := typDPT);
STLV59_563.STLV59_A_563_212.RB601_V := M1_096_212_RB601_V.xSwitch_OUT;
M1_097_212_RB601_HVAC(bPortKNX := 1, dwIndex_DPT := 97, typDPT := typDPT);
STLV59_563.STLV59_A_563_212.RB601_HVAC := M1_097_212_RB601_HVAC.xSwitch_OUT;
(* RT601_CT *)
(* RT602_CT *)
M1_098_212_RT601_CT(bPortKNX := 1, dwIndex_DPT := 98, typDPT := typDPT);
STLV59_563.STLV59_A_563_212.RT601_CT := M1_098_212_RT601_CT.rValue_OUT;
M1_099_212_RT602_CT(bPortKNX := 1, dwIndex_DPT := 99, typDPT := typDPT);
STLV59_563.STLV59_A_563_212.RT602_CT := M1_099_212_RT602_CT.rValue_OUT;
(* RY601_CV *)
M1_100_212_RY601_CV(bPortKNX := 1, dwIndex_DPT := 100, typDPT := typDPT);
STLV59_563.STLV59_A_563_212.RY601_CV := M1_100_212_RY601_CV.rValue_OUT;
(* Rom 213 *)
(* RB601_V *)
(* RB601_HVAC *)
M1_101_213_RB601_V(bPortKNX := 1, dwIndex_DPT := 101, typDPT := typDPT);
STLV59_563.STLV59_A_563_213.RB601_V := M1_101_213_RB601_V.xSwitch_OUT;
M1_102_213_RB601_HVAC(bPortKNX := 1, dwIndex_DPT := 102, typDPT := typDPT);
STLV59_563.STLV59_A_563_213.RB601_HVAC := M1_102_213_RB601_HVAC.xSwitch_OUT;
(* RT601_CT *)
(* RT602_CT *)
M1_103_213_RT601_CT(bPortKNX := 1, dwIndex_DPT := 103, typDPT := typDPT);
STLV59_563.STLV59_A_563_213.RT601_CT := M1_103_213_RT601_CT.rValue_OUT;
M1_104_213_RT602_CT(bPortKNX := 1, dwIndex_DPT := 104, typDPT := typDPT);
STLV59_563.STLV59_A_563_213.RT602_CT := M1_104_213_RT602_CT.rValue_OUT;
(* Rom T1_U1 *)
(* RB601_V *)
(* RB601_HVAC *)
M1_105_T1_U1_RB601_V(bPortKNX := 1, dwIndex_DPT := 105, typDPT := typDPT);
STLV59_563.STLV59_A_563_T1_U1.RB601_V := M1_105_T1_U1_RB601_V.xSwitch_OUT;
M1_106_T1_U1_RB601_HVAC(bPortKNX := 1, dwIndex_DPT := 106, typDPT := typDPT);
STLV59_563.STLV59_A_563_T1_U1.RB601_HVAC := M1_106_T1_U1_RB601_HVAC.xSwitch_OUT;
(* RT601_CT *)
(* RT602_CT *)
M1_107_T1_U1_RT601_CT(bPortKNX := 1, dwIndex_DPT := 107, typDPT := typDPT);
STLV59_563.STLV59_A_563_T1_U1.RT601_CT := M1_107_T1_U1_RT601_CT.rValue_OUT;
M1_108_T1_U1_RT602_CT(bPortKNX := 1, dwIndex_DPT := 108, typDPT := typDPT);
STLV59_563.STLV59_A_563_T1_U1.RT602_CT := M1_108_T1_U1_RT602_CT.rValue_OUT;
(* Rom T2_1 *)
(* RB601_V *)
(* RB601_HVAC *)
M1_109_T2_1_RB601_V(bPortKNX := 1, dwIndex_DPT := 109, typDPT := typDPT);
STLV59_563.STLV59_A_563_T2_1.RB601_V := M1_109_T2_1_RB601_V.xSwitch_OUT;
M1_110_T2_1_RB601_HVAC(bPortKNX := 1, dwIndex_DPT := 110, typDPT := typDPT);
STLV59_563.STLV59_A_563_T2_1.RB601_HVAC := M1_110_T2_1_RB601_HVAC.xSwitch_OUT;
(* RT601_CT *)
(* RT602_CT *)
M1_111_T2_1_RT601_CT(bPortKNX := 1, dwIndex_DPT := 111, typDPT := typDPT);
STLV59_563.STLV59_A_563_T2_1.RT601_CT := M1_111_T2_1_RT601_CT.rValue_OUT;
M1_112_T2_1_RT602_CT(bPortKNX := 1, dwIndex_DPT := 112, typDPT := typDPT);
STLV59_563.STLV59_A_563_T2_1.RT602_CT := M1_112_T2_1_RT602_CT.rValue_OUT;
(* Rom T2_2 *)
(* RB601_V *)
(* RB601_HVAC *)
M1_113_T2_2_RB601_V(bPortKNX := 1, dwIndex_DPT := 113, typDPT := typDPT);
STLV59_563.STLV59_A_563_T2_2.RB601_V := M1_113_T2_2_RB601_V.xSwitch_OUT;
M1_114_T2_2_RB601_HVAC(bPortKNX := 1, dwIndex_DPT := 114, typDPT := typDPT);
STLV59_563.STLV59_A_563_T2_2.RB601_HVAC := M1_114_T2_2_RB601_HVAC.xSwitch_OUT;
(* RT601_CT *)
(* RT602_CT *)
M1_115_T2_2_RT601_CT(bPortKNX := 1, dwIndex_DPT := 115, typDPT := typDPT);
STLV59_563.STLV59_A_563_T2_2.RT601_CT := M1_115_T2_2_RT601_CT.rValue_OUT;
M1_116_T2_2_RT602_CT(bPortKNX := 1, dwIndex_DPT := 116, typDPT := typDPT);
STLV59_563.STLV59_A_563_T2_2.RT602_CT := M1_116_T2_2_RT602_CT.rValue_OUT;
END_PROGRAM

PROGRAM PRG_563_Romstyring
  VAR
    Rom_001 : fbRomtype_22200000221102;  (* 001 *)
    Rom_002 : fbRomtype_1120011;  (* 002 *)
    Rom_003 : fbRomtype_112001;  (* 003 *)
    Rom_004 : fbRomtype_112101;  (* 004 *)
    Rom_005 : fbRomtype_112001;  (* 005 *)
    Rom_006 : fbRomtype_112002;  (* 006 *)
    Rom_007 : fbRomtype_112001;  (* 007 *)
    Rom_008 : fbRomtype_112001;  (* 008 *)
    Rom_009 : fbRomtype_112001;  (* 009 *)
    Rom_010 : fbRomtype_112001;  (* 010 *)
    Rom_011 : fbRomtype_112001;  (* 011 *)
    Rom_012 : fbRomtype_112001;  (* 012 *)
    Rom_013 : fbRomtype_112001;  (* 013 *)
    Rom_017 : fbRomtype_112001;  (* 017 *)
    Rom_101 : fbRomtype_112001;  (* 101 *)
    Rom_102 : fbRomtype_112001;  (* 102 *)
    Rom_103 : fbRomtype_4462051;  (* 103 *)
    Rom_109 : fbRomtype_112001;  (* 109 *)
    Rom_212 : fbRomtype_1121011;  (* 212 *)
    Rom_213 : fbRomtype_1120011;  (* 213 *)
    Rom_T1_U1 : fbRomtype_112001;  (* T1_U1 *)
    Rom_T2_1 : fbRomtype_112001;  (* T2_1 *)
    Rom_T2_2 : fbRomtype_112001;  (* T2_2 *)
  END_VAR

(* CFC diagram, written out as Structured Text *)
(* Rom 001 *)
Rom_001(RB601_HVAC := STLV59_563.STLV59_A_563_001.RB601_HVAC, RB602_HVAC := STLV59_563.STLV59_A_563_001.RB602_HVAC, RT601_CT := STLV59_563.STLV59_A_563_001.RT601_CT, RT602_CT := STLV59_563.STLV59_A_563_001.RT602_CT, RT602_SP := STLV59_563.STLV59_A_563_001.RT602_SP, RT601_SP_D := STLV59_563.STLV59_A_563_001.RT601_SP_D, RT601_SP_S := STLV59_563.STLV59_A_563_001.RT601_SP_S, RT601_SP_N := STLV59_563.STLV59_A_563_001.RT601_SP_N, RT601_SP_F := STLV59_563.STLV59_A_563_001.RT601_SP_F, OPM := STLV59_563.STLV59_A_563_001.OPM, RT601_SP_IN := STLV59_563.STLV59_A_563_001.RT601_SP_IN, RT602_SP_IN := STLV59_563.STLV59_A_563_001.RT602_SP_IN, LU601_V := STLV59_563.STLV59_A_563_001.LU601_V);
STLV59_563.STLV59_A_563_001.OPM_CV := Rom_001.OPM_CV;
STLV59_563.STLV59_A_563_001.RT601_CS := Rom_001.RT601_CS;
STLV59_563.STLV59_A_563_001.OPM_001 := Rom_001.OPM_001;
STLV59_563.STLV59_A_563_001.OPM_002 := Rom_001.OPM_002;
(* Rom 002 *)
Rom_002(RB601_HVAC := STLV59_563.STLV59_A_563_002.RB601_HVAC, RT601_CT := STLV59_563.STLV59_A_563_002.RT601_CT, RT602_CT := STLV59_563.STLV59_A_563_002.RT602_CT, RT602_SP := STLV59_563.STLV59_A_563_002.RT602_SP, RT601_SP_D := STLV59_563.STLV59_A_563_002.RT601_SP_D, RT601_SP_S := STLV59_563.STLV59_A_563_002.RT601_SP_S, RT601_SP_N := STLV59_563.STLV59_A_563_002.RT601_SP_N, RT601_SP_F := STLV59_563.STLV59_A_563_002.RT601_SP_F, OPM := STLV59_563.STLV59_A_563_002.OPM, LH601_MAN := STLV59_563.STLV59_A_563_002.LH601_MAN, LC601_SP := STLV59_563.STLV59_A_563_002.LC601_SP, LC601_MAN := STLV59_563.STLV59_A_563_002.LC601_MAN);
STLV59_563.STLV59_A_563_002.OPM_CV := Rom_002.OPM_CV;
STLV59_563.STLV59_A_563_002.RT601_CS := Rom_002.RT601_CS;
STLV59_563.STLV59_A_563_002.LH601_CMD := Rom_002.LH601_CMD;
STLV59_563.STLV59_A_563_002.LC601_OP := Rom_002.LC601_OP;
(* Rom 003 *)
Rom_003(RB601_HVAC := STLV59_563.STLV59_A_563_003.RB601_HVAC, RT601_CT := STLV59_563.STLV59_A_563_003.RT601_CT, RT602_CT := STLV59_563.STLV59_A_563_003.RT602_CT, RT602_SP := STLV59_563.STLV59_A_563_003.RT602_SP, RT601_SP_D := STLV59_563.STLV59_A_563_003.RT601_SP_D, RT601_SP_S := STLV59_563.STLV59_A_563_003.RT601_SP_S, RT601_SP_N := STLV59_563.STLV59_A_563_003.RT601_SP_N, RT601_SP_F := STLV59_563.STLV59_A_563_003.RT601_SP_F, OPM := STLV59_563.STLV59_A_563_003.OPM, LH601_MAN := STLV59_563.STLV59_A_563_003.LH601_MAN);
STLV59_563.STLV59_A_563_003.OPM_CV := Rom_003.OPM_CV;
STLV59_563.STLV59_A_563_003.RT601_CS := Rom_003.RT601_CS;
STLV59_563.STLV59_A_563_003.LH601_CMD := Rom_003.LH601_CMD;
(* Rom 004 *)
Rom_004(RB601_HVAC := STLV59_563.STLV59_A_563_004.RB601_HVAC, RT601_CT := STLV59_563.STLV59_A_563_004.RT601_CT, RT602_CT := STLV59_563.STLV59_A_563_004.RT602_CT, RT602_SP := STLV59_563.STLV59_A_563_004.RT602_SP, RT601_SP_D := STLV59_563.STLV59_A_563_004.RT601_SP_D, RT601_SP_S := STLV59_563.STLV59_A_563_004.RT601_SP_S, RT601_SP_N := STLV59_563.STLV59_A_563_004.RT601_SP_N, RT601_SP_F := STLV59_563.STLV59_A_563_004.RT601_SP_F, OPM := STLV59_563.STLV59_A_563_004.OPM, RY601_CV := STLV59_563.STLV59_A_563_004.RY601_CV, RY601_SP := STLV59_563.STLV59_A_563_004.RY601_SP, LH601_MAN := STLV59_563.STLV59_A_563_004.LH601_MAN);
STLV59_563.STLV59_A_563_004.OPM_CV := Rom_004.OPM_CV;
STLV59_563.STLV59_A_563_004.RT601_CS := Rom_004.RT601_CS;
STLV59_563.STLV59_A_563_004.RY601_OP := Rom_004.RY601_OP;
STLV59_563.STLV59_A_563_004.LH601_CMD := Rom_004.LH601_CMD;
(* Rom 005 *)
Rom_005(RB601_HVAC := STLV59_563.STLV59_A_563_005.RB601_HVAC, RT601_CT := STLV59_563.STLV59_A_563_005.RT601_CT, RT602_CT := STLV59_563.STLV59_A_563_005.RT602_CT, RT602_SP := STLV59_563.STLV59_A_563_005.RT602_SP, RT601_SP_D := STLV59_563.STLV59_A_563_005.RT601_SP_D, RT601_SP_S := STLV59_563.STLV59_A_563_005.RT601_SP_S, RT601_SP_N := STLV59_563.STLV59_A_563_005.RT601_SP_N, RT601_SP_F := STLV59_563.STLV59_A_563_005.RT601_SP_F, OPM := STLV59_563.STLV59_A_563_005.OPM, LH601_MAN := STLV59_563.STLV59_A_563_005.LH601_MAN);
STLV59_563.STLV59_A_563_005.OPM_CV := Rom_005.OPM_CV;
STLV59_563.STLV59_A_563_005.RT601_CS := Rom_005.RT601_CS;
STLV59_563.STLV59_A_563_005.LH601_CMD := Rom_005.LH601_CMD;
(* Rom 006 *)
Rom_006(RB601_HVAC := STLV59_563.STLV59_A_563_006.RB601_HVAC, RT601_CT := STLV59_563.STLV59_A_563_006.RT601_CT, RT602_CT := STLV59_563.STLV59_A_563_006.RT602_CT, RT602_SP := STLV59_563.STLV59_A_563_006.RT602_SP, RT601_SP_D := STLV59_563.STLV59_A_563_006.RT601_SP_D, RT601_SP_S := STLV59_563.STLV59_A_563_006.RT601_SP_S, RT601_SP_N := STLV59_563.STLV59_A_563_006.RT601_SP_N, RT601_SP_F := STLV59_563.STLV59_A_563_006.RT601_SP_F, OPM := STLV59_563.STLV59_A_563_006.OPM, LH601_MAN := STLV59_563.STLV59_A_563_006.LH601_MAN);
STLV59_563.STLV59_A_563_006.OPM_CV := Rom_006.OPM_CV;
STLV59_563.STLV59_A_563_006.RT601_CS := Rom_006.RT601_CS;
STLV59_563.STLV59_A_563_006.LH601_CMD := Rom_006.LH601_CMD;
STLV59_563.STLV59_A_563_006.LH602_CMD := Rom_006.LH602_CMD;
(* Rom 007 *)
Rom_007(RB601_HVAC := STLV59_563.STLV59_A_563_007.RB601_HVAC, RT601_CT := STLV59_563.STLV59_A_563_007.RT601_CT, RT602_CT := STLV59_563.STLV59_A_563_007.RT602_CT, RT602_SP := STLV59_563.STLV59_A_563_007.RT602_SP, RT601_SP_D := STLV59_563.STLV59_A_563_007.RT601_SP_D, RT601_SP_S := STLV59_563.STLV59_A_563_007.RT601_SP_S, RT601_SP_N := STLV59_563.STLV59_A_563_007.RT601_SP_N, RT601_SP_F := STLV59_563.STLV59_A_563_007.RT601_SP_F, OPM := STLV59_563.STLV59_A_563_007.OPM, LH601_MAN := STLV59_563.STLV59_A_563_007.LH601_MAN);
STLV59_563.STLV59_A_563_007.OPM_CV := Rom_007.OPM_CV;
STLV59_563.STLV59_A_563_007.RT601_CS := Rom_007.RT601_CS;
STLV59_563.STLV59_A_563_007.LH601_CMD := Rom_007.LH601_CMD;
(* Rom 008 *)
Rom_008(RB601_HVAC := STLV59_563.STLV59_A_563_008.RB601_HVAC, RT601_CT := STLV59_563.STLV59_A_563_008.RT601_CT, RT602_CT := STLV59_563.STLV59_A_563_008.RT602_CT, RT602_SP := STLV59_563.STLV59_A_563_008.RT602_SP, RT601_SP_D := STLV59_563.STLV59_A_563_008.RT601_SP_D, RT601_SP_S := STLV59_563.STLV59_A_563_008.RT601_SP_S, RT601_SP_N := STLV59_563.STLV59_A_563_008.RT601_SP_N, RT601_SP_F := STLV59_563.STLV59_A_563_008.RT601_SP_F, OPM := STLV59_563.STLV59_A_563_008.OPM, LH601_MAN := STLV59_563.STLV59_A_563_008.LH601_MAN);
STLV59_563.STLV59_A_563_008.OPM_CV := Rom_008.OPM_CV;
STLV59_563.STLV59_A_563_008.RT601_CS := Rom_008.RT601_CS;
STLV59_563.STLV59_A_563_008.LH601_CMD := Rom_008.LH601_CMD;
(* Rom 009 *)
Rom_009(RB601_HVAC := STLV59_563.STLV59_A_563_009.RB601_HVAC, RT601_CT := STLV59_563.STLV59_A_563_009.RT601_CT, RT602_CT := STLV59_563.STLV59_A_563_009.RT602_CT, RT602_SP := STLV59_563.STLV59_A_563_009.RT602_SP, RT601_SP_D := STLV59_563.STLV59_A_563_009.RT601_SP_D, RT601_SP_S := STLV59_563.STLV59_A_563_009.RT601_SP_S, RT601_SP_N := STLV59_563.STLV59_A_563_009.RT601_SP_N, RT601_SP_F := STLV59_563.STLV59_A_563_009.RT601_SP_F, OPM := STLV59_563.STLV59_A_563_009.OPM, LH601_MAN := STLV59_563.STLV59_A_563_009.LH601_MAN);
STLV59_563.STLV59_A_563_009.OPM_CV := Rom_009.OPM_CV;
STLV59_563.STLV59_A_563_009.RT601_CS := Rom_009.RT601_CS;
STLV59_563.STLV59_A_563_009.LH601_CMD := Rom_009.LH601_CMD;
(* Rom 010 *)
Rom_010(RB601_HVAC := STLV59_563.STLV59_A_563_010.RB601_HVAC, RT601_CT := STLV59_563.STLV59_A_563_010.RT601_CT, RT602_CT := STLV59_563.STLV59_A_563_010.RT602_CT, RT602_SP := STLV59_563.STLV59_A_563_010.RT602_SP, RT601_SP_D := STLV59_563.STLV59_A_563_010.RT601_SP_D, RT601_SP_S := STLV59_563.STLV59_A_563_010.RT601_SP_S, RT601_SP_N := STLV59_563.STLV59_A_563_010.RT601_SP_N, RT601_SP_F := STLV59_563.STLV59_A_563_010.RT601_SP_F, OPM := STLV59_563.STLV59_A_563_010.OPM, LH601_MAN := STLV59_563.STLV59_A_563_010.LH601_MAN);
STLV59_563.STLV59_A_563_010.OPM_CV := Rom_010.OPM_CV;
STLV59_563.STLV59_A_563_010.RT601_CS := Rom_010.RT601_CS;
STLV59_563.STLV59_A_563_010.LH601_CMD := Rom_010.LH601_CMD;
(* Rom 011 *)
Rom_011(RB601_HVAC := STLV59_563.STLV59_A_563_011.RB601_HVAC, RT601_CT := STLV59_563.STLV59_A_563_011.RT601_CT, RT602_CT := STLV59_563.STLV59_A_563_011.RT602_CT, RT602_SP := STLV59_563.STLV59_A_563_011.RT602_SP, RT601_SP_D := STLV59_563.STLV59_A_563_011.RT601_SP_D, RT601_SP_S := STLV59_563.STLV59_A_563_011.RT601_SP_S, RT601_SP_N := STLV59_563.STLV59_A_563_011.RT601_SP_N, RT601_SP_F := STLV59_563.STLV59_A_563_011.RT601_SP_F, OPM := STLV59_563.STLV59_A_563_011.OPM, LH601_MAN := STLV59_563.STLV59_A_563_011.LH601_MAN);
STLV59_563.STLV59_A_563_011.OPM_CV := Rom_011.OPM_CV;
STLV59_563.STLV59_A_563_011.RT601_CS := Rom_011.RT601_CS;
STLV59_563.STLV59_A_563_011.LH601_CMD := Rom_011.LH601_CMD;
(* Rom 012 *)
Rom_012(RB601_HVAC := STLV59_563.STLV59_A_563_012.RB601_HVAC, RT601_CT := STLV59_563.STLV59_A_563_012.RT601_CT, RT602_CT := STLV59_563.STLV59_A_563_012.RT602_CT, RT602_SP := STLV59_563.STLV59_A_563_012.RT602_SP, RT601_SP_D := STLV59_563.STLV59_A_563_012.RT601_SP_D, RT601_SP_S := STLV59_563.STLV59_A_563_012.RT601_SP_S, RT601_SP_N := STLV59_563.STLV59_A_563_012.RT601_SP_N, RT601_SP_F := STLV59_563.STLV59_A_563_012.RT601_SP_F, OPM := STLV59_563.STLV59_A_563_012.OPM, LH601_MAN := STLV59_563.STLV59_A_563_012.LH601_MAN);
STLV59_563.STLV59_A_563_012.OPM_CV := Rom_012.OPM_CV;
STLV59_563.STLV59_A_563_012.RT601_CS := Rom_012.RT601_CS;
STLV59_563.STLV59_A_563_012.LH601_CMD := Rom_012.LH601_CMD;
(* Rom 013 *)
Rom_013(RB601_HVAC := STLV59_563.STLV59_A_563_013.RB601_HVAC, RT601_CT := STLV59_563.STLV59_A_563_013.RT601_CT, RT602_CT := STLV59_563.STLV59_A_563_013.RT602_CT, RT602_SP := STLV59_563.STLV59_A_563_013.RT602_SP, RT601_SP_D := STLV59_563.STLV59_A_563_013.RT601_SP_D, RT601_SP_S := STLV59_563.STLV59_A_563_013.RT601_SP_S, RT601_SP_N := STLV59_563.STLV59_A_563_013.RT601_SP_N, RT601_SP_F := STLV59_563.STLV59_A_563_013.RT601_SP_F, OPM := STLV59_563.STLV59_A_563_013.OPM, LH601_MAN := STLV59_563.STLV59_A_563_013.LH601_MAN);
STLV59_563.STLV59_A_563_013.OPM_CV := Rom_013.OPM_CV;
STLV59_563.STLV59_A_563_013.RT601_CS := Rom_013.RT601_CS;
STLV59_563.STLV59_A_563_013.LH601_CMD := Rom_013.LH601_CMD;
(* Rom 017 *)
Rom_017(RB601_HVAC := STLV59_563.STLV59_A_563_017.RB601_HVAC, RT601_CT := STLV59_563.STLV59_A_563_017.RT601_CT, RT602_CT := STLV59_563.STLV59_A_563_017.RT602_CT, RT602_SP := STLV59_563.STLV59_A_563_017.RT602_SP, RT601_SP_D := STLV59_563.STLV59_A_563_017.RT601_SP_D, RT601_SP_S := STLV59_563.STLV59_A_563_017.RT601_SP_S, RT601_SP_N := STLV59_563.STLV59_A_563_017.RT601_SP_N, RT601_SP_F := STLV59_563.STLV59_A_563_017.RT601_SP_F, OPM := STLV59_563.STLV59_A_563_017.OPM, LH601_MAN := STLV59_563.STLV59_A_563_017.LH601_MAN);
STLV59_563.STLV59_A_563_017.OPM_CV := Rom_017.OPM_CV;
STLV59_563.STLV59_A_563_017.RT601_CS := Rom_017.RT601_CS;
STLV59_563.STLV59_A_563_017.LH601_CMD := Rom_017.LH601_CMD;
(* Rom 101 *)
Rom_101(RB601_HVAC := STLV59_563.STLV59_A_563_101.RB601_HVAC, RT601_CT := STLV59_563.STLV59_A_563_101.RT601_CT, RT602_CT := STLV59_563.STLV59_A_563_101.RT602_CT, RT602_SP := STLV59_563.STLV59_A_563_101.RT602_SP, RT601_SP_D := STLV59_563.STLV59_A_563_101.RT601_SP_D, RT601_SP_S := STLV59_563.STLV59_A_563_101.RT601_SP_S, RT601_SP_N := STLV59_563.STLV59_A_563_101.RT601_SP_N, RT601_SP_F := STLV59_563.STLV59_A_563_101.RT601_SP_F, OPM := STLV59_563.STLV59_A_563_101.OPM, LH601_MAN := STLV59_563.STLV59_A_563_101.LH601_MAN);
STLV59_563.STLV59_A_563_101.OPM_CV := Rom_101.OPM_CV;
STLV59_563.STLV59_A_563_101.RT601_CS := Rom_101.RT601_CS;
STLV59_563.STLV59_A_563_101.LH601_CMD := Rom_101.LH601_CMD;
(* Rom 102 *)
Rom_102(RB601_HVAC := STLV59_563.STLV59_A_563_102.RB601_HVAC, RT601_CT := STLV59_563.STLV59_A_563_102.RT601_CT, RT602_CT := STLV59_563.STLV59_A_563_102.RT602_CT, RT602_SP := STLV59_563.STLV59_A_563_102.RT602_SP, RT601_SP_D := STLV59_563.STLV59_A_563_102.RT601_SP_D, RT601_SP_S := STLV59_563.STLV59_A_563_102.RT601_SP_S, RT601_SP_N := STLV59_563.STLV59_A_563_102.RT601_SP_N, RT601_SP_F := STLV59_563.STLV59_A_563_102.RT601_SP_F, OPM := STLV59_563.STLV59_A_563_102.OPM, LH601_MAN := STLV59_563.STLV59_A_563_102.LH601_MAN);
STLV59_563.STLV59_A_563_102.OPM_CV := Rom_102.OPM_CV;
STLV59_563.STLV59_A_563_102.RT601_CS := Rom_102.RT601_CS;
STLV59_563.STLV59_A_563_102.LH601_CMD := Rom_102.LH601_CMD;
(* Rom 103 *)
Rom_103(RB601_HVAC := STLV59_563.STLV59_A_563_103.RB601_HVAC, RB602_HVAC := STLV59_563.STLV59_A_563_103.RB602_HVAC, RB603_HVAC := STLV59_563.STLV59_A_563_103.RB603_HVAC, RB604_HVAC := STLV59_563.STLV59_A_563_103.RB604_HVAC, RT601_CT := STLV59_563.STLV59_A_563_103.RT601_CT, RT602_CT := STLV59_563.STLV59_A_563_103.RT602_CT, RT602_SP := STLV59_563.STLV59_A_563_103.RT602_SP, RT603_CT := STLV59_563.STLV59_A_563_103.RT603_CT, RT603_SP := STLV59_563.STLV59_A_563_103.RT603_SP, RT604_CT := STLV59_563.STLV59_A_563_103.RT604_CT, RT604_SP := STLV59_563.STLV59_A_563_103.RT604_SP, RT605_CT := STLV59_563.STLV59_A_563_103.RT605_CT, RT605_SP := STLV59_563.STLV59_A_563_103.RT605_SP, RT606_CT := STLV59_563.STLV59_A_563_103.RT606_CT, RT606_SP := STLV59_563.STLV59_A_563_103.RT606_SP, RT601_SP_D := STLV59_563.STLV59_A_563_103.RT601_SP_D, RT601_SP_S := STLV59_563.STLV59_A_563_103.RT601_SP_S, RT601_SP_N := STLV59_563.STLV59_A_563_103.RT601_SP_N, RT601_SP_F := STLV59_563.STLV59_A_563_103.RT601_SP_F, OPM := STLV59_563.STLV59_A_563_103.OPM, RY601_CV := STLV59_563.STLV59_A_563_103.RY601_CV, RY602_CV := STLV59_563.STLV59_A_563_103.RY602_CV, RY601_SP := STLV59_563.STLV59_A_563_103.RY601_SP, LH601_MAN := STLV59_563.STLV59_A_563_103.LH601_MAN, LC601_SP := STLV59_563.STLV59_A_563_103.LC601_SP, LC601_MAN := STLV59_563.STLV59_A_563_103.LC601_MAN);
STLV59_563.STLV59_A_563_103.OPM_CV := Rom_103.OPM_CV;
STLV59_563.STLV59_A_563_103.RT601_CS := Rom_103.RT601_CS;
STLV59_563.STLV59_A_563_103.RY601_OP := Rom_103.RY601_OP;
STLV59_563.STLV59_A_563_103.LH601_CMD := Rom_103.LH601_CMD;
STLV59_563.STLV59_A_563_103.LH602_CMD := Rom_103.LH602_CMD;
STLV59_563.STLV59_A_563_103.LH603_CMD := Rom_103.LH603_CMD;
STLV59_563.STLV59_A_563_103.LH604_CMD := Rom_103.LH604_CMD;
STLV59_563.STLV59_A_563_103.LH605_CMD := Rom_103.LH605_CMD;
STLV59_563.STLV59_A_563_103.LC601_OP := Rom_103.LC601_OP;
(* Rom 109 *)
Rom_109(RB601_HVAC := STLV59_563.STLV59_A_563_109.RB601_HVAC, RT601_CT := STLV59_563.STLV59_A_563_109.RT601_CT, RT602_CT := STLV59_563.STLV59_A_563_109.RT602_CT, RT602_SP := STLV59_563.STLV59_A_563_109.RT602_SP, RT601_SP_D := STLV59_563.STLV59_A_563_109.RT601_SP_D, RT601_SP_S := STLV59_563.STLV59_A_563_109.RT601_SP_S, RT601_SP_N := STLV59_563.STLV59_A_563_109.RT601_SP_N, RT601_SP_F := STLV59_563.STLV59_A_563_109.RT601_SP_F, OPM := STLV59_563.STLV59_A_563_109.OPM, LH601_MAN := STLV59_563.STLV59_A_563_109.LH601_MAN);
STLV59_563.STLV59_A_563_109.OPM_CV := Rom_109.OPM_CV;
STLV59_563.STLV59_A_563_109.RT601_CS := Rom_109.RT601_CS;
STLV59_563.STLV59_A_563_109.LH601_CMD := Rom_109.LH601_CMD;
(* Rom 212 *)
Rom_212(RB601_HVAC := STLV59_563.STLV59_A_563_212.RB601_HVAC, RT601_CT := STLV59_563.STLV59_A_563_212.RT601_CT, RT602_CT := STLV59_563.STLV59_A_563_212.RT602_CT, RT602_SP := STLV59_563.STLV59_A_563_212.RT602_SP, RT601_SP_D := STLV59_563.STLV59_A_563_212.RT601_SP_D, RT601_SP_S := STLV59_563.STLV59_A_563_212.RT601_SP_S, RT601_SP_N := STLV59_563.STLV59_A_563_212.RT601_SP_N, RT601_SP_F := STLV59_563.STLV59_A_563_212.RT601_SP_F, OPM := STLV59_563.STLV59_A_563_212.OPM, RY601_CV := STLV59_563.STLV59_A_563_212.RY601_CV, RY601_SP := STLV59_563.STLV59_A_563_212.RY601_SP, LH601_MAN := STLV59_563.STLV59_A_563_212.LH601_MAN, LC601_SP := STLV59_563.STLV59_A_563_212.LC601_SP, LC601_MAN := STLV59_563.STLV59_A_563_212.LC601_MAN);
STLV59_563.STLV59_A_563_212.OPM_CV := Rom_212.OPM_CV;
STLV59_563.STLV59_A_563_212.RT601_CS := Rom_212.RT601_CS;
STLV59_563.STLV59_A_563_212.RY601_OP := Rom_212.RY601_OP;
STLV59_563.STLV59_A_563_212.LH601_CMD := Rom_212.LH601_CMD;
STLV59_563.STLV59_A_563_212.LC601_OP := Rom_212.LC601_OP;
(* Rom 213 *)
Rom_213(RB601_HVAC := STLV59_563.STLV59_A_563_213.RB601_HVAC, RT601_CT := STLV59_563.STLV59_A_563_213.RT601_CT, RT602_CT := STLV59_563.STLV59_A_563_213.RT602_CT, RT602_SP := STLV59_563.STLV59_A_563_213.RT602_SP, RT601_SP_D := STLV59_563.STLV59_A_563_213.RT601_SP_D, RT601_SP_S := STLV59_563.STLV59_A_563_213.RT601_SP_S, RT601_SP_N := STLV59_563.STLV59_A_563_213.RT601_SP_N, RT601_SP_F := STLV59_563.STLV59_A_563_213.RT601_SP_F, OPM := STLV59_563.STLV59_A_563_213.OPM, LH601_MAN := STLV59_563.STLV59_A_563_213.LH601_MAN, LC601_SP := STLV59_563.STLV59_A_563_213.LC601_SP, LC601_MAN := STLV59_563.STLV59_A_563_213.LC601_MAN);
STLV59_563.STLV59_A_563_213.OPM_CV := Rom_213.OPM_CV;
STLV59_563.STLV59_A_563_213.RT601_CS := Rom_213.RT601_CS;
STLV59_563.STLV59_A_563_213.LH601_CMD := Rom_213.LH601_CMD;
STLV59_563.STLV59_A_563_213.LC601_OP := Rom_213.LC601_OP;
(* Rom T1_U1 *)
Rom_T1_U1(RB601_HVAC := STLV59_563.STLV59_A_563_T1_U1.RB601_HVAC, RT601_CT := STLV59_563.STLV59_A_563_T1_U1.RT601_CT, RT602_CT := STLV59_563.STLV59_A_563_T1_U1.RT602_CT, RT602_SP := STLV59_563.STLV59_A_563_T1_U1.RT602_SP, RT601_SP_D := STLV59_563.STLV59_A_563_T1_U1.RT601_SP_D, RT601_SP_S := STLV59_563.STLV59_A_563_T1_U1.RT601_SP_S, RT601_SP_N := STLV59_563.STLV59_A_563_T1_U1.RT601_SP_N, RT601_SP_F := STLV59_563.STLV59_A_563_T1_U1.RT601_SP_F, OPM := STLV59_563.STLV59_A_563_T1_U1.OPM, LH601_MAN := STLV59_563.STLV59_A_563_T1_U1.LH601_MAN);
STLV59_563.STLV59_A_563_T1_U1.OPM_CV := Rom_T1_U1.OPM_CV;
STLV59_563.STLV59_A_563_T1_U1.RT601_CS := Rom_T1_U1.RT601_CS;
STLV59_563.STLV59_A_563_T1_U1.LH601_CMD := Rom_T1_U1.LH601_CMD;
(* Rom T2_1 *)
Rom_T2_1(RB601_HVAC := STLV59_563.STLV59_A_563_T2_1.RB601_HVAC, RT601_CT := STLV59_563.STLV59_A_563_T2_1.RT601_CT, RT602_CT := STLV59_563.STLV59_A_563_T2_1.RT602_CT, RT602_SP := STLV59_563.STLV59_A_563_T2_1.RT602_SP, RT601_SP_D := STLV59_563.STLV59_A_563_T2_1.RT601_SP_D, RT601_SP_S := STLV59_563.STLV59_A_563_T2_1.RT601_SP_S, RT601_SP_N := STLV59_563.STLV59_A_563_T2_1.RT601_SP_N, RT601_SP_F := STLV59_563.STLV59_A_563_T2_1.RT601_SP_F, OPM := STLV59_563.STLV59_A_563_T2_1.OPM, LH601_MAN := STLV59_563.STLV59_A_563_T2_1.LH601_MAN);
STLV59_563.STLV59_A_563_T2_1.OPM_CV := Rom_T2_1.OPM_CV;
STLV59_563.STLV59_A_563_T2_1.RT601_CS := Rom_T2_1.RT601_CS;
STLV59_563.STLV59_A_563_T2_1.LH601_CMD := Rom_T2_1.LH601_CMD;
(* Rom T2_2 *)
Rom_T2_2(RB601_HVAC := STLV59_563.STLV59_A_563_T2_2.RB601_HVAC, RT601_CT := STLV59_563.STLV59_A_563_T2_2.RT601_CT, RT602_CT := STLV59_563.STLV59_A_563_T2_2.RT602_CT, RT602_SP := STLV59_563.STLV59_A_563_T2_2.RT602_SP, RT601_SP_D := STLV59_563.STLV59_A_563_T2_2.RT601_SP_D, RT601_SP_S := STLV59_563.STLV59_A_563_T2_2.RT601_SP_S, RT601_SP_N := STLV59_563.STLV59_A_563_T2_2.RT601_SP_N, RT601_SP_F := STLV59_563.STLV59_A_563_T2_2.RT601_SP_F, OPM := STLV59_563.STLV59_A_563_T2_2.OPM, LH601_MAN := STLV59_563.STLV59_A_563_T2_2.LH601_MAN);
STLV59_563.STLV59_A_563_T2_2.OPM_CV := Rom_T2_2.OPM_CV;
STLV59_563.STLV59_A_563_T2_2.RT601_CS := Rom_T2_2.RT601_CS;
STLV59_563.STLV59_A_563_T2_2.LH601_CMD := Rom_T2_2.LH601_CMD;
END_PROGRAM

PROGRAM PRG_360_HVAC

	STLV59_563.STLV59_A_563_RB001_HVAC:=
(
	STLV59_563.STLV59_A_563_001.RB601_HVAC OR
	STLV59_563.STLV59_A_563_001.RB602_HVAC OR
	STLV59_563.STLV59_A_563_002.RB601_HVAC OR
	STLV59_563.STLV59_A_563_003.RB601_HVAC OR
	STLV59_563.STLV59_A_563_004.RB601_HVAC OR
	STLV59_563.STLV59_A_563_005.RB601_HVAC OR
	STLV59_563.STLV59_A_563_006.RB601_HVAC OR
	STLV59_563.STLV59_A_563_007.RB601_HVAC OR
	STLV59_563.STLV59_A_563_008.RB601_HVAC OR
	STLV59_563.STLV59_A_563_009.RB601_HVAC OR
	STLV59_563.STLV59_A_563_010.RB601_HVAC OR
	STLV59_563.STLV59_A_563_011.RB601_HVAC OR
	STLV59_563.STLV59_A_563_012.RB601_HVAC OR
	STLV59_563.STLV59_A_563_013.RB601_HVAC OR
	STLV59_563.STLV59_A_563_014.RB601_HVAC OR
	STLV59_563.STLV59_A_563_014.RB602_HVAC OR
	STLV59_563.STLV59_A_563_015.RB601_HVAC OR
	STLV59_563.STLV59_A_563_016.RB601_HVAC OR
	STLV59_563.STLV59_A_563_017.RB601_HVAC OR
	STLV59_563.STLV59_A_563_101.RB601_HVAC OR
	STLV59_563.STLV59_A_563_102.RB601_HVAC OR
	STLV59_563.STLV59_A_563_103.RB601_HVAC OR
	STLV59_563.STLV59_A_563_103.RB602_HVAC OR
	STLV59_563.STLV59_A_563_103.RB603_HVAC OR
	STLV59_563.STLV59_A_563_103.RB604_HVAC OR
	STLV59_563.STLV59_A_563_109.RB601_HVAC OR
	STLV59_563.STLV59_A_563_212.RB601_HVAC OR
	STLV59_563.STLV59_A_563_213.RB601_HVAC OR
	STLV59_563.STLV59_A_563_T1_U1.RB601_HVAC OR
	STLV59_563.STLV59_A_563_T2_1.RB601_HVAC OR
	STLV59_563.STLV59_A_563_T2_2.RB601_HVAC
);
END_PROGRAM
